// TIA Portal V15.1 export
// export: Created 2024-06-21T08:40:54.0593079Z, ExportSetting WithDefaults, DisplayName Totally Integrated Automation Portal, DisplayVersion V15.1 Update 5, DisplayName TIA Portal Openness, DisplayVersion V15.1 Update 5, DisplayName SINAMICS Startdrive Advanced, DisplayVersion V15.1, DisplayName G130, G150, S120, S150, SINAMICS MV, S210, DisplayVersion V15.1, DisplayName G110M, G120, G120C, G120D, G120P, DisplayVersion V15.1, DisplayName STEP 7 Professional, DisplayVersion V15.1 Update 5, DisplayName STEP 7 Safety, DisplayVersion V15.1, DisplayName WinCC Professional, DisplayVersion V15.1 Update 5, DisplayName SIMATIC Visualization Architect, DisplayVersion V15.1
FUNCTION "LDWordToBit" : Void   // FC1014, FBD
TITLE = LDWordToBit
{ S7_Optimized_Access := 'TRUE' }
AUTHOR : VCC
FAMILY : Control
NAME : DWor2Bit
VERSION : 0.1
// =============================================================================
// Moves One Double Word to 32 bits 
// =============================================================================
// stored: AutoNumber false, IsIECCheckEnabled false, SetENOAutomatically False, UDAEnableTagReadback false
   VAR_INPUT
      I_DWord : DWord;   // Input DWord
   END_VAR
   VAR_OUTPUT
      O_0 : Bool;   // Output 0
      O_1 : Bool;   // Output 1
      O_2 : Bool;   // Output 2
      O_3 : Bool;   // Output 3
      O_4 : Bool;   // Output 4
      O_5 : Bool;   // Output 5
      O_6 : Bool;   // Output 6
      O_7 : Bool;   // Output 7
      O_8 : Bool;   // Output 8
      O_9 : Bool;   // Output 9
      O_10 : Bool;   // Output 10
      O_11 : Bool;   // Output 11
      O_12 : Bool;   // Output 12
      O_13 : Bool;   // Output 13
      O_14 : Bool;   // Output 14
      O_15 : Bool;   // Output 15
      O_16 : Bool;   // Output 16
      O_17 : Bool;   // Output 17
      O_18 : Bool;   // Output 18
      O_19 : Bool;   // Output 19
      O_20 : Bool;   // Output 20
      O_21 : Bool;   // Output 21
      O_22 : Bool;   // Output 22
      O_23 : Bool;   // Output 23
      O_24 : Bool;   // Output 24
      O_25 : Bool;   // Output 25
      O_26 : Bool;   // Output 26
      O_27 : Bool;   // Output 27
      O_28 : Bool;   // Output 28
      O_29 : Bool;   // Output 29
      O_30 : Bool;   // Output 30
      O_31 : Bool;   // Output 31
   END_VAR
BEGIN

REGION Network 1: **** 8 - Outputs **** Bit from temporary Word to output
   // Copy bit 0 from temporary Word to output
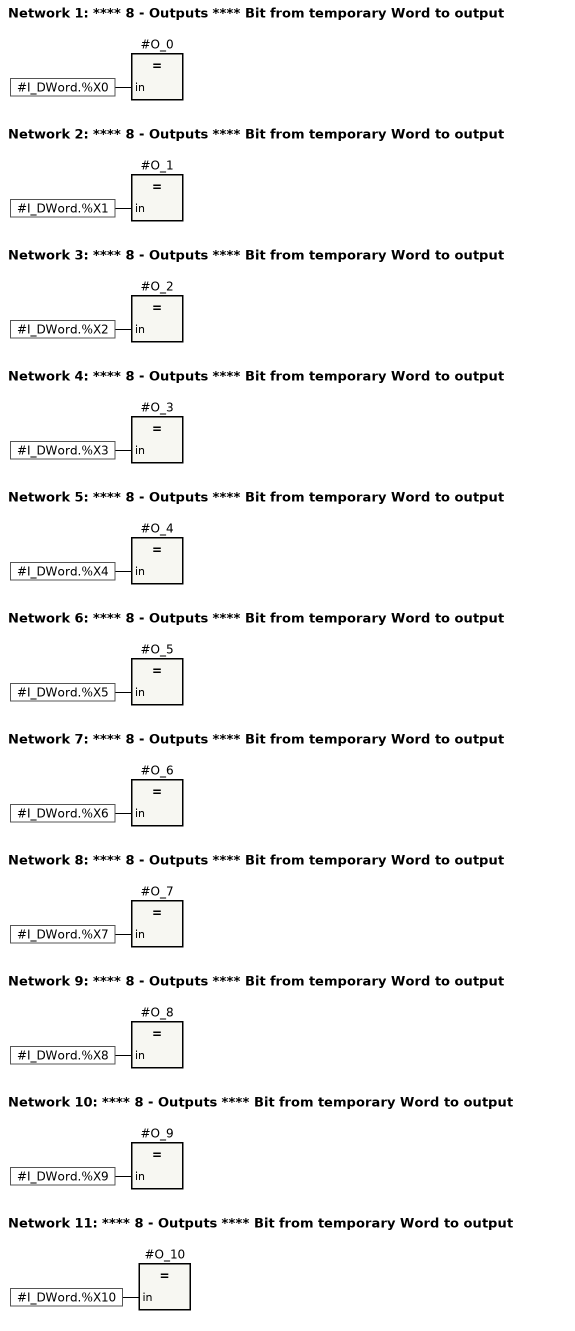
   #O_0 := #I_DWord.%X0;
END_REGION

REGION Network 2: **** 8 - Outputs **** Bit from temporary Word to output
   // Copy bit 1 from temporary Word to output
   #O_1 := #I_DWord.%X1;
END_REGION

REGION Network 3: **** 8 - Outputs **** Bit from temporary Word to output
   // Copy bit 2 from temporary Word to output
   #O_2 := #I_DWord.%X2;
END_REGION

REGION Network 4: **** 8 - Outputs **** Bit from temporary Word to output
   // Copy bit 3 from temporary Word to output
   #O_3 := #I_DWord.%X3;
END_REGION

REGION Network 5: **** 8 - Outputs **** Bit from temporary Word to output
   // Copy bit 4 from temporary Word to output
   #O_4 := #I_DWord.%X4;
END_REGION

REGION Network 6: **** 8 - Outputs **** Bit from temporary Word to output
   // Copy bit 5 from temporary Word to output
   #O_5 := #I_DWord.%X5;
END_REGION

REGION Network 7: **** 8 - Outputs **** Bit from temporary Word to output
   // Copy bit 6 from temporary Word to output
   #O_6 := #I_DWord.%X6;
END_REGION

REGION Network 8: **** 8 - Outputs **** Bit from temporary Word to output
   // Copy bit 7 from temporary Word to output
   #O_7 := #I_DWord.%X7;
END_REGION

REGION Network 9: **** 8 - Outputs **** Bit from temporary Word to output
   // Copy bit 8 from temporary Word to output
   #O_8 := #I_DWord.%X8;
END_REGION

REGION Network 10: **** 8 - Outputs **** Bit from temporary Word to output
   // Copy bit 9 from temporary Word to output
   #O_9 := #I_DWord.%X9;
END_REGION

REGION Network 11: **** 8 - Outputs **** Bit from temporary Word to output
   // Copy bit 10 from temporary Word to output
   #O_10 := #I_DWord.%X10;
END_REGION

REGION Network 12: **** 8 - Outputs **** Bit from temporary Word to output
   // Copy bit 11 from temporary Word to output
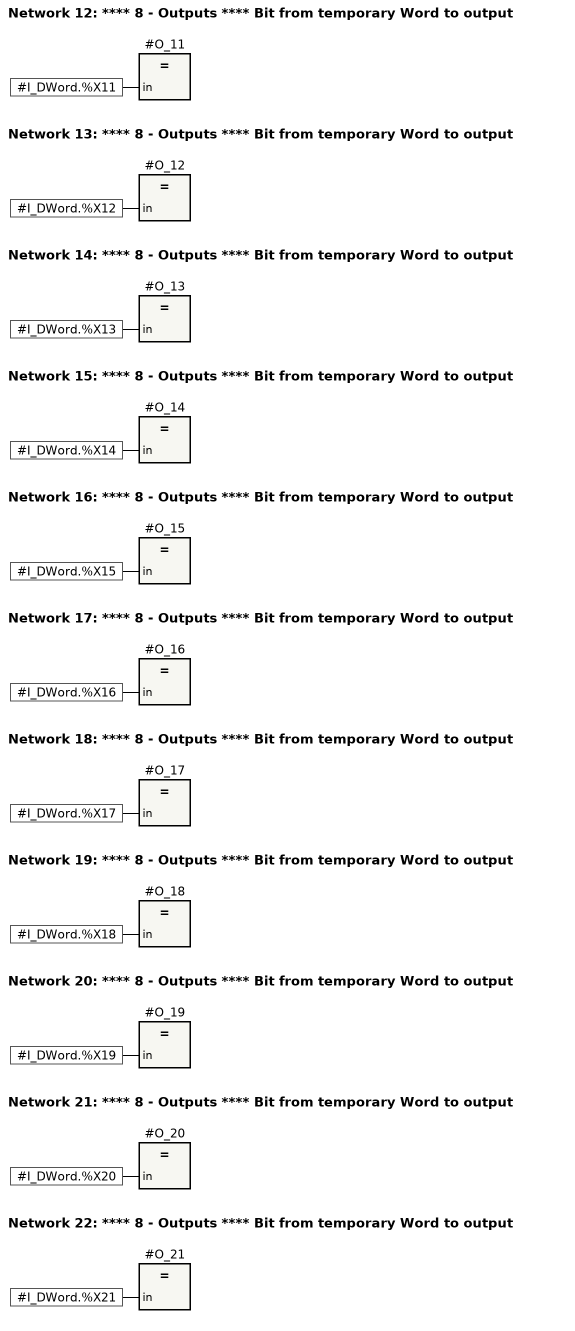
   #O_11 := #I_DWord.%X11;
END_REGION

REGION Network 13: **** 8 - Outputs **** Bit from temporary Word to output
   // Copy bit 12 from temporary Word to output
   #O_12 := #I_DWord.%X12;
END_REGION

REGION Network 14: **** 8 - Outputs **** Bit from temporary Word to output
   // Copy bit 13 from temporary Word to output
   #O_13 := #I_DWord.%X13;
END_REGION

REGION Network 15: **** 8 - Outputs **** Bit from temporary Word to output
   // Copy bit 14 from temporary Word to output
   #O_14 := #I_DWord.%X14;
END_REGION

REGION Network 16: **** 8 - Outputs **** Bit from temporary Word to output
   // Copy bit 15 from temporary Word to output
   #O_15 := #I_DWord.%X15;
END_REGION

REGION Network 17: **** 8 - Outputs **** Bit from temporary Word to output
   // Copy bit 16 from temporary Word to output
   #O_16 := #I_DWord.%X16;
END_REGION

REGION Network 18: **** 8 - Outputs **** Bit from temporary Word to output
   // Copy bit 17 from temporary Word to output
   #O_17 := #I_DWord.%X17;
END_REGION

REGION Network 19: **** 8 - Outputs **** Bit from temporary Word to output
   // Copy bit 18 from temporary Word to output
   #O_18 := #I_DWord.%X18;
END_REGION

REGION Network 20: **** 8 - Outputs **** Bit from temporary Word to output
   // Copy bit 19 from temporary Word to output
   #O_19 := #I_DWord.%X19;
END_REGION

REGION Network 21: **** 8 - Outputs **** Bit from temporary Word to output
   // Copy bit 20 from temporary Word to output
   #O_20 := #I_DWord.%X20;
END_REGION

REGION Network 22: **** 8 - Outputs **** Bit from temporary Word to output
   // Copy bit 21 from temporary Word to output
   #O_21 := #I_DWord.%X21;
END_REGION

REGION Network 23: **** 8 - Outputs **** Bit from temporary Word to output
   // Copy bit 22 from temporary Word to output
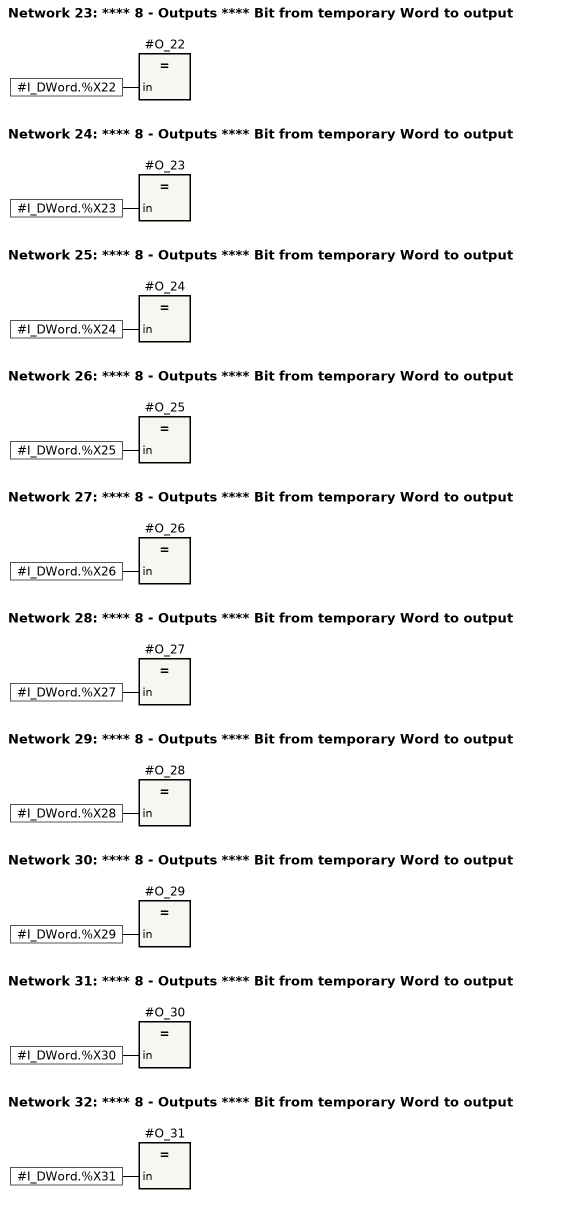
   #O_22 := #I_DWord.%X22;
END_REGION

REGION Network 24: **** 8 - Outputs **** Bit from temporary Word to output
   // Copy bit 23 from temporary Word to output
   #O_23 := #I_DWord.%X23;
END_REGION

REGION Network 25: **** 8 - Outputs **** Bit from temporary Word to output
   // Copy bit 24 from temporary Word to output
   #O_24 := #I_DWord.%X24;
END_REGION

REGION Network 26: **** 8 - Outputs **** Bit from temporary Word to output
   // Copy bit 25 from temporary Word to output
   #O_25 := #I_DWord.%X25;
END_REGION

REGION Network 27: **** 8 - Outputs **** Bit from temporary Word to output
   // Copy bit 26 from temporary Word to output
   #O_26 := #I_DWord.%X26;
END_REGION

REGION Network 28: **** 8 - Outputs **** Bit from temporary Word to output
   // Copy bit 27 from temporary Word to output
   #O_27 := #I_DWord.%X27;
END_REGION

REGION Network 29: **** 8 - Outputs **** Bit from temporary Word to output
   // Copy bit 28 from temporary Word to output
   #O_28 := #I_DWord.%X28;
END_REGION

REGION Network 30: **** 8 - Outputs **** Bit from temporary Word to output
   // Copy bit 29 from temporary Word to output
   #O_29 := #I_DWord.%X29;
END_REGION

REGION Network 31: **** 8 - Outputs **** Bit from temporary Word to output
   // Copy bit 30 from temporary Word to output
   #O_30 := #I_DWord.%X30;
END_REGION

REGION Network 32: **** 8 - Outputs **** Bit from temporary Word to output
   // Copy bit 31 from temporary Word to output
   #O_31 := #I_DWord.%X31;
END_REGION
END_FUNCTION
